Fanuc KAREL source: kt00191.KL

PROGRAM KT00191
%STACKSIZE=65535
%PRIORITY=65535
%NOLOCKGROUP
VAR
OUT : INTEGER
-- UNRESOLVED DECLARATIONS (source type spelling not recovered)
-- H1 : ARRAY[2] OF TYPE_0x0017 (type_u16=0x2017)
-- H2 : ARRAY[2] OF TYPE_0x0017 (type_u16=0x2017)
BEGIN
-- UNRESOLVED_PC line 8 opcodes [2E 22 9D 33 B4] marker_code=0
-- UNRESOLVED_PC line 9 opcodes [2E 22 9D 33 B4] marker_code=19
-- UNRESOLVED_PC line 10 opcodes [2E 22 9D 33 B4] marker_code=38
-- UNRESOLVED_PC line 11 opcodes [2E 22 9D 33 B4] marker_code=57
-- UNRESOLVED_PC line 12 opcodes [22 9D 33 B3 22 9D 33 B3 56 23] marker_code=76
END KT00191
